PROGRAM PRG_TEST
VAR
	fbGantryAutoCoupling_Test : FB_GantryAutoCoupling_Test;
END_VAR

TcUnit.RUN();

END_PROGRAM

(* stored: Version 1.1.0.1, ProductVersion 3.1.4022.12
   POU PRG_TEST: Id {fdb013bd-9e82-4044-94c0-4ed8f18460f5}, SpecialFunc None *)
